(* Logix 5000 project; controller cal1632 1756-L62 rev 16.20; software revision 16.05; part 26 of 61 *)
(* tags used below, declared in another part *)
   AFI : BOOL;
   FAULT : BOOL;
   p01_param_turret_dia_ft : REAL;
   p01r02 : routine;
   p01r09_pb_global_reset : BOOL;
   p01r12_selected_line_speed : REAL;
   p01r13_line_running : BOOL;
   p01r13_line_slow_ramp : BOOL;
   p02_dint_from_hmi : hmi_dint;
   p11r31_timer_prs : TIMER;
   p13r03_hz : SYS_SCP;
   p13r30_request_cool : BOOL;
   p19_ai_prs : REAL;
   p19_di_pump : BOOL;
   p19_do_pump : BOOL;
   p19_param_zone_pressure : REAL;
   p19r30_request_cool : BOOL;
   p19r31 : routine;
   p19r31_pb_start : BOOL;
   p19r31_pb_stop : BOOL;
   p19r31_request_a00 : BOOL;
   p19r31_request_auto_run : BOOL;
   p19r31_request_manual_run : BOOL;
   p19r31_run_permissive : BOOL;
   p19r31_timer_fault : TIMER[4];
   p19r31_timer_warning : TIMER[4];
   p20_acc_fill_time_sec : REAL;
   p20_acc_input_max : REAL;
   p20_acc_input_min : REAL;
   p20_acc_output_max : REAL;
   p20_acc_output_min : REAL;
   p20_ai_acc_pstn : REAL;
   p20_ai_lc01 : REAL;
   p20_ai_letoff_dia : REAL;
   p20_ai_lo_turret_amps : REAL;
   p20_ai_lo_turret_hz : REAL;
   p20_ai_lo_turret_speed : REAL;
   p20_ai_loa_speed : REAL;
   p20_ai_lob_speed : REAL;
   p20_di_acc_door_open : BOOL;
   p20_di_acc_empty : BOOL;
   p20_di_acc_full : BOOL;
   p20_di_clutch_prs_ok : BOOL;
   p20_di_lfr_jog_fwd : BOOL;
   p20_di_lfr_jog_rev : BOOL;
   p20_di_lfr_nip_close : BOOL;
   p20_di_lo_turret : acs800_di_normal;
   p20_di_lo_turret_therm : BOOL;
   p20_di_loa_active : BOOL;
   p20_di_loa_brake : BOOL;
   p20_di_loa_fwd_dir : BOOL;
   p20_di_loa_jog : BOOL;
   p20_di_loa_start : BOOL;
   p20_di_loa_stop : BOOL;
   p20_di_loa_temp : BOOL;
   p20_di_lob_brake_thermostat : BOOL;
   p20_di_lob_fwd_dir : BOOL;
   p20_di_lob_jog : BOOL;
   p20_di_lob_motor_thermostat : BOOL;
   p20_di_lob_start : BOOL;
   p20_di_lob_stop : BOOL;
   p20_di_lof_acc_fill : BOOL;
   p20_di_turret_fwd : BOOL;
   p20_di_turret_pos : BOOL;
   p20_di_turret_rev : BOOL;
   p20_dia_input_max : REAL;
   p20_dia_input_min : REAL;
   p20_dia_output_max : REAL;
   p20_dia_output_min : REAL;
   p20_dint_to_hmi : DINT[16];
   p20_lc_input_max : REAL;
   p20_lc_input_min : REAL;
   p20_lc_output_max : REAL;
   p20_lc_output_min : REAL;
   p20_loa_ai_amps : REAL;
   p20_loa_ai_hz : REAL;
   p20_loa_ai_rpm : REAL;
   p20_loa_ai_torque : REAL;
   p20_loa_footage_input_max : REAL;
   p20_loa_footage_input_min : REAL;
   p20_loa_footage_output_max : REAL;
   p20_loa_footage_output_min : REAL;
   p20_lob_ai_amps : REAL;
   p20_lob_ai_hz : REAL;
   p20_lob_ai_rpm : REAL;
   p20_lob_ai_torque : REAL;
   p20_lob_footage_input_max : REAL;
   p20_lob_footage_input_min : REAL;
   p20_lob_footage_output_max : REAL;
   p20_lob_footage_output_min : REAL;
   p20_param_lo_turret_gear_ratio : REAL;
   p20_param_loa_gear_ratio : REAL;
   p20_param_lob_gear_ratio : REAL;
   p20_vfd_di_loa : acs800_di_normal;
   p20_vfd_di_lob : acs800_di_normal;
   p20r01 : routine;
   p20r02 : routine;
   p20r02_fault_exists : BOOL;
   p20r02_letoff_dia_ft : REAL;
   p20r02_letoff_selection_dwell : TIMER;
   p20r02_timer_fault : TIMER[4];
   p20r02_timer_warning : TIMER[4];
   p20r02_unack_fault : BOOL;
   p20r02_unack_warning : BOOL;
   p20r02_warning_exists : BOOL;
   p20r03 : routine;
   p20r03_accumulator_pct_scp : SYS_SCP;
   p20r03_accumulator_scp : SYS_SCP;
   p20r03_distance_to_core : REAL;
   p20r03_lo_radius : REAL;
   p20r03_lo_turret_speed_fb : SYS_RPM_TO_SPEED;
   p20r03_loa_distance_to_core : REAL;
   p20r03_Loa_footage_scp : SYS_SCP;
   p20r03_loa_speed_fb : SYS_RPM_TO_SPEED;
   p20r03_load_cell : SYS_SCP;
   p20r03_lob_distance_to_core : REAL;
   p20r03_Lob_footage_scp : SYS_SCP;
   p20r03_lob_speed_fb : SYS_RPM_TO_SPEED;
   p20r03_sensor_input : REAL;
   p20r03_sensor_scp : SYS_SCP;
   p20r03_timer_fault : TIMER[4];
   p20r03_timer_warning : TIMER[4];
   p20r04 : routine;
   p20r05 : routine;
   p20r06 : routine;
   p20r07 : routine;
   p20r08 : routine;
   p20r09 : routine;
   p20r10 : routine;
   p20r11 : routine;
   p20r13 : routine;
   p20r13_ai_acc_pct : REAL;
   p20r13_ai_loa_footage_ft : REAL;
   p20r13_ai_lob_footage_ft : REAL;
   p20r14 : routine;
   p20r15 : routine;
   p20r15_loa_on : BOOL;
   p20r16 : routine;
   p20r16_lob_on : BOOL;
   p20r17 : routine;
   p20r17_letoff_avg_diam_inch : REAL;
   p20r18 : routine;
   p22_ao_selected_speed : REAL;
(* P19_Advanced_Cooling, continued *)

ROUTINE R31_Pump   (* ladder *)
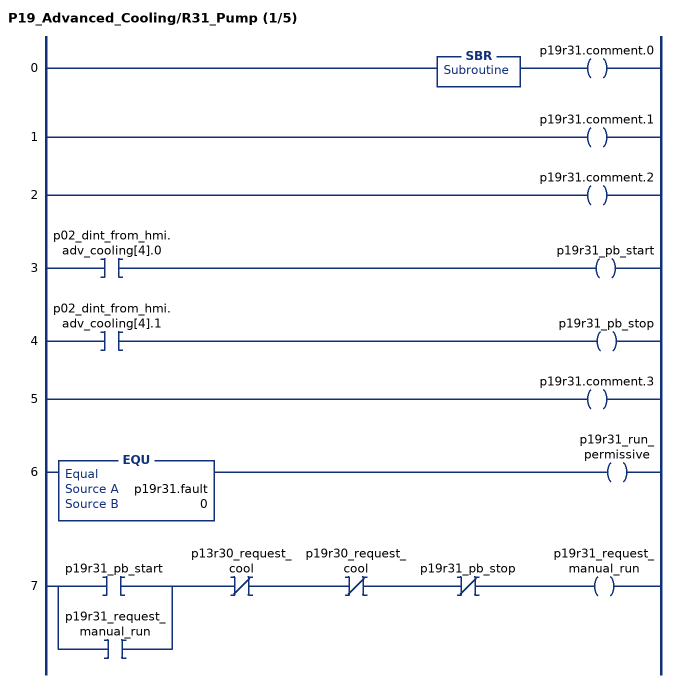
   0: SBR()OTE(p19r31.comment.0);
   1: OTE(p19r31.comment.1);
   2: OTE(p19r31.comment.2);
   3: XIC(p02_dint_from_hmi.adv_cooling[4].0)OTE(p19r31_pb_start);
   4: XIC(p02_dint_from_hmi.adv_cooling[4].1)OTE(p19r31_pb_stop);
   5: OTE(p19r31.comment.3);
   6: EQU(p19r31.fault,0)OTE(p19r31_run_permissive);
   7: [XIC(p19r31_pb_start) ,XIC(p19r31_request_manual_run) ]XIO(p13r30_request_cool)XIO(p19r30_request_cool)XIO(p19r31_pb_stop)OTE(p19r31_request_manual_run);
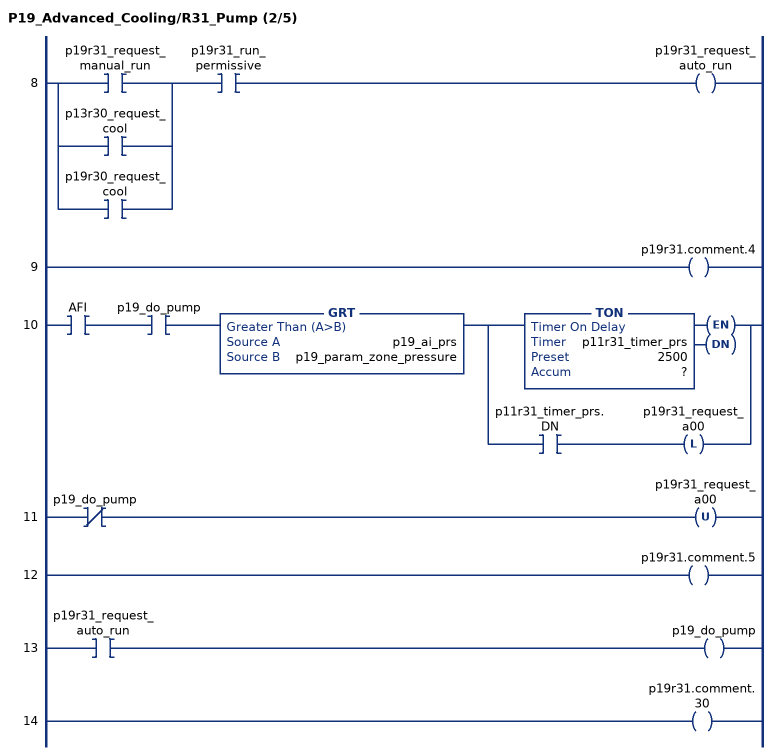
   8: [XIC(p19r31_request_manual_run) ,XIC(p13r30_request_cool) ,XIC(p19r30_request_cool) ]XIC(p19r31_run_permissive)OTE(p19r31_request_auto_run);
   9: OTE(p19r31.comment.4);
   10: XIC(AFI)XIC(p19_do_pump)GRT(p19_ai_prs,p19_param_zone_pressure)[TON(p11r31_timer_prs,?,?) ,XIC(p11r31_timer_prs.DN) OTL(p19r31_request_a00) ];
   11: XIO(p19_do_pump)OTU(p19r31_request_a00);
   12: OTE(p19r31.comment.5);
   13: XIC(p19r31_request_auto_run)OTE(p19_do_pump);
   14: OTE(p19r31.comment.30);
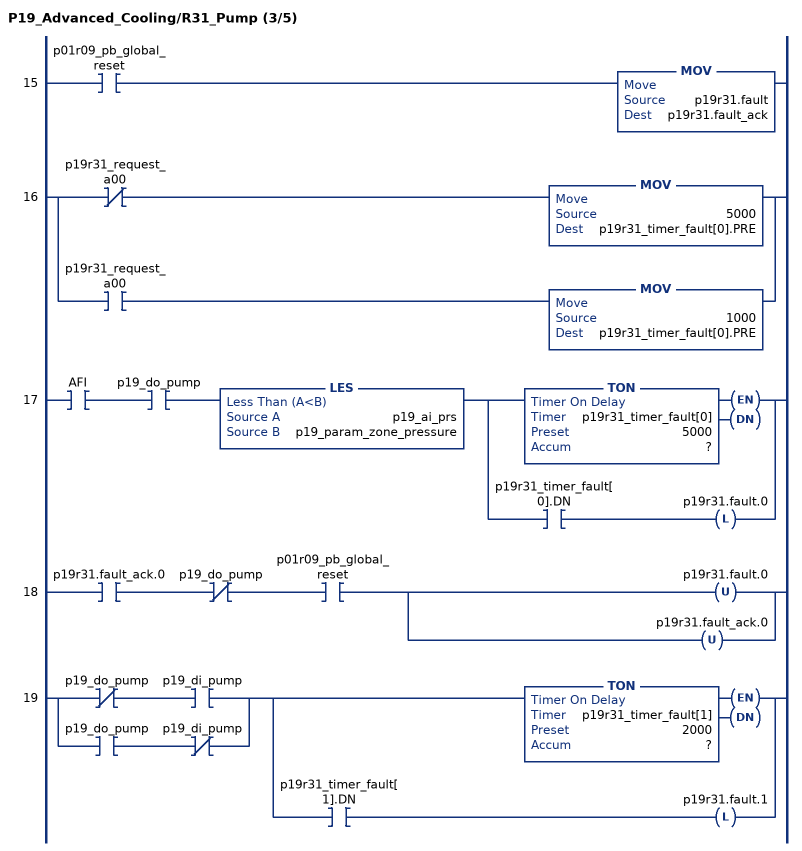
   15: XIC(p01r09_pb_global_reset)MOV(p19r31.fault,p19r31.fault_ack);
   16: [XIO(p19r31_request_a00) MOV(5000,p19r31_timer_fault[0].PRE) ,XIC(p19r31_request_a00) MOV(1000,p19r31_timer_fault[0].PRE) ];
   17: XIC(AFI)XIC(p19_do_pump)LES(p19_ai_prs,p19_param_zone_pressure)[TON(p19r31_timer_fault[0],?,?) ,XIC(p19r31_timer_fault[0].DN) OTL(p19r31.fault.0) ];
   18: XIC(p19r31.fault_ack.0)XIO(p19_do_pump)XIC(p01r09_pb_global_reset)[OTU(p19r31.fault.0) ,OTU(p19r31.fault_ack.0) ];
   19: [XIO(p19_do_pump) XIC(p19_di_pump) ,XIC(p19_do_pump) XIO(p19_di_pump) ][TON(p19r31_timer_fault[1],?,?) ,XIC(p19r31_timer_fault[1].DN) OTL(p19r31.fault.1) ];
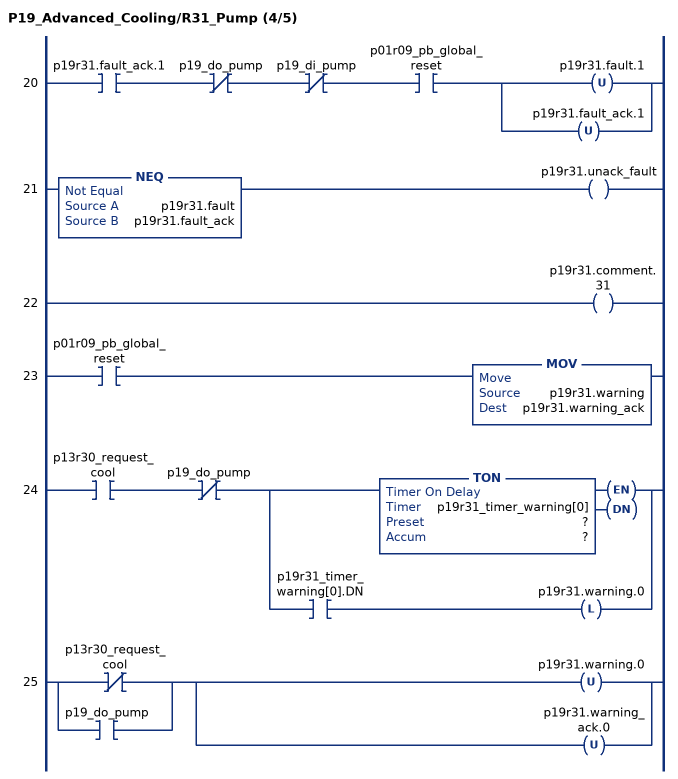
   20: XIC(p19r31.fault_ack.1)XIO(p19_do_pump)XIO(p19_di_pump)XIC(p01r09_pb_global_reset)[OTU(p19r31.fault.1) ,OTU(p19r31.fault_ack.1) ];
   21: NEQ(p19r31.fault,p19r31.fault_ack)OTE(p19r31.unack_fault);
   22: OTE(p19r31.comment.31);
   23: XIC(p01r09_pb_global_reset)MOV(p19r31.warning,p19r31.warning_ack);
   24: XIC(p13r30_request_cool)XIO(p19_do_pump)[TON(p19r31_timer_warning[0],?,?) ,XIC(p19r31_timer_warning[0].DN) OTL(p19r31.warning.0) ];
   25: [XIO(p13r30_request_cool) ,XIC(p19_do_pump) ][OTU(p19r31.warning.0) ,OTU(p19r31.warning_ack.0) ];
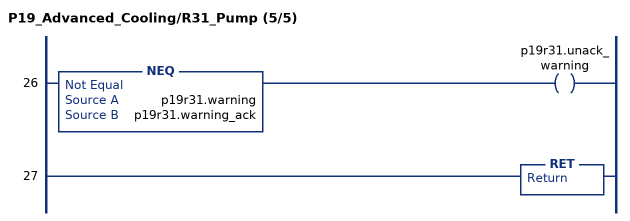
   26: NEQ(p19r31.warning,p19r31.warning_ack)OTE(p19r31.unack_warning);
   27: RET();
END_ROUTINE
END_PROGRAM

PROGRAM P20_Letoff   (* main routine R01_Main *)

ROUTINE R01_Main   (* ladder *)
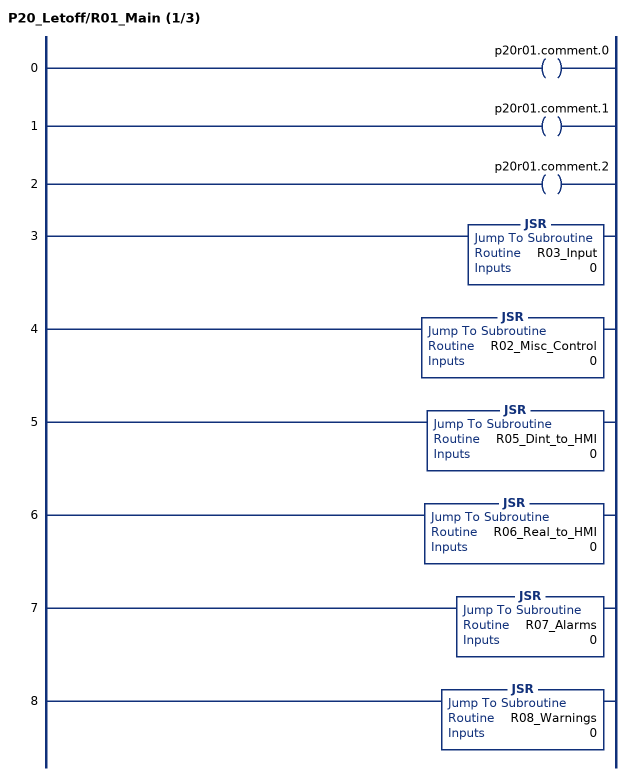
   0: OTE(p20r01.comment.0);
   1: OTE(p20r01.comment.1);
   2: OTE(p20r01.comment.2);
   3: JSR(R03_Input,0);
   4: JSR(R02_Misc_Control,0);
   5: JSR(R05_Dint_to_HMI,0);
   6: JSR(R06_Real_to_HMI,0);
   7: JSR(R07_Alarms,0);
   8: JSR(R08_Warnings,0);
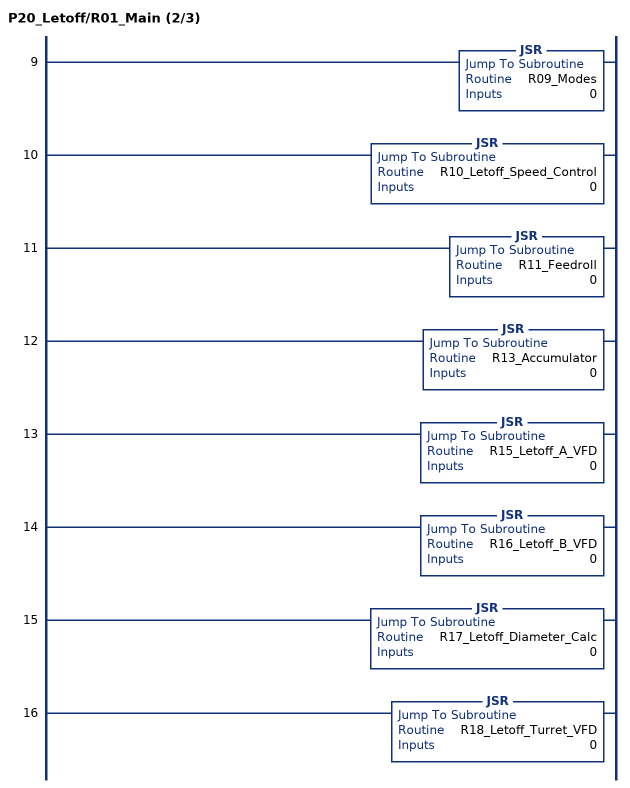
   9: JSR(R09_Modes,0);
   10: JSR(R10_Letoff_Speed_Control,0);
   11: JSR(R11_Feedroll,0);
   12: JSR(R13_Accumulator,0);
   13: JSR(R15_Letoff_A_VFD,0);
   14: JSR(R16_Letoff_B_VFD,0);
   15: JSR(R17_Letoff_Diameter_Calc,0);
   16: JSR(R18_Letoff_Turret_VFD,0);
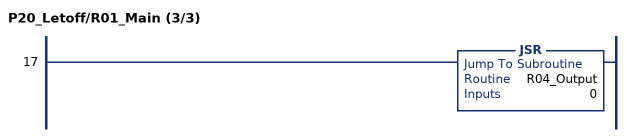
   17: JSR(R04_Output,0);
END_ROUTINE

ROUTINE R02_Misc_Control   (* ladder *)
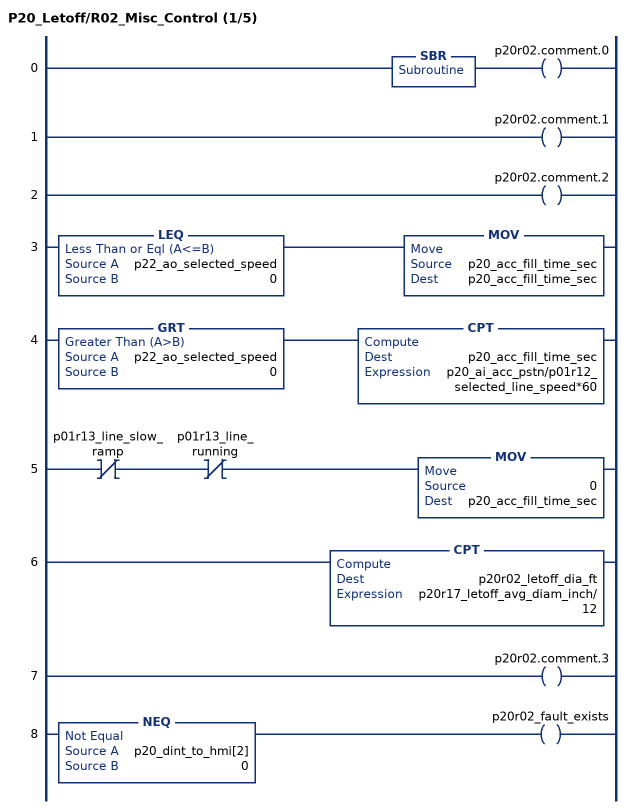
   0: SBR()OTE(p20r02.comment.0);
   1: OTE(p20r02.comment.1);
   2: OTE(p20r02.comment.2);
   3: LEQ(p22_ao_selected_speed,0)MOV(p20_acc_fill_time_sec,p20_acc_fill_time_sec);
   4: GRT(p22_ao_selected_speed,0)CPT(p20_acc_fill_time_sec,p20_ai_acc_pstn/p01r12_selected_line_speed*60);
   5: XIO(p01r13_line_slow_ramp)XIO(p01r13_line_running)MOV(0,p20_acc_fill_time_sec);
   6: CPT(p20r02_letoff_dia_ft,p20r17_letoff_avg_diam_inch/12);
   7: OTE(p20r02.comment.3);
   8: NEQ(p20_dint_to_hmi[2],0)OTE(p20r02_fault_exists);
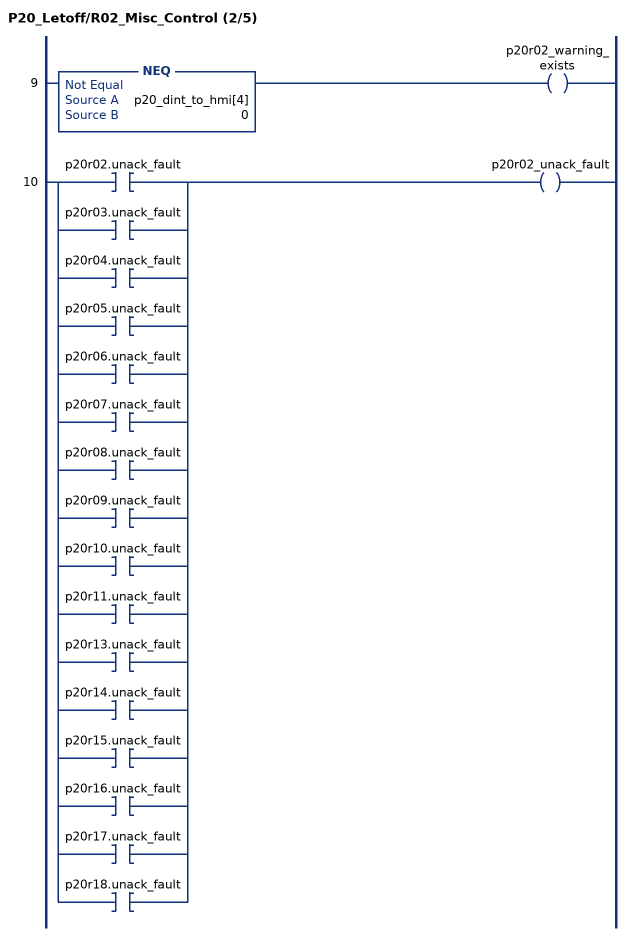
   9: NEQ(p20_dint_to_hmi[4],0)OTE(p20r02_warning_exists);
   10: [XIC(p20r02.unack_fault) ,XIC(p20r03.unack_fault) ,XIC(p20r04.unack_fault) ,XIC(p20r05.unack_fault) ,XIC(p20r06.unack_fault) ,XIC(p20r07.unack_fault) ,XIC(p20r08.unack_fault) ,XIC(p20r09.unack_fault) ,XIC(p20r10.unack_fault) ,XIC(p20r11.unack_fault) ,XIC(p20r13.unack_fault) ,XIC(p20r14.unack_fault) ,XIC(p20r15.unack_fault) ,XIC(p20r16.unack_fault) ,XIC(p20r17.unack_fault) ,XIC(p20r18.unack_fault) ]OTE(p20r02_unack_fault);
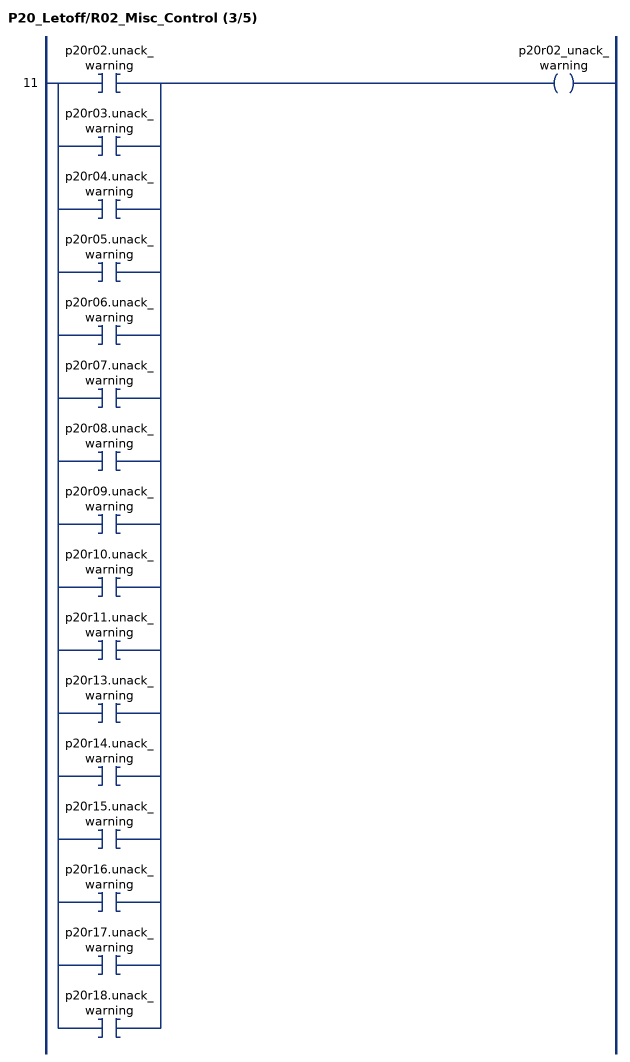
   11: [XIC(p20r02.unack_warning) ,XIC(p20r03.unack_warning) ,XIC(p20r04.unack_warning) ,XIC(p20r05.unack_warning) ,XIC(p20r06.unack_warning) ,XIC(p20r07.unack_warning) ,XIC(p20r08.unack_warning) ,XIC(p20r09.unack_warning) ,XIC(p20r10.unack_warning) ,XIC(p20r11.unack_warning) ,XIC(p20r13.unack_warning) ,XIC(p20r14.unack_warning) ,XIC(p20r15.unack_warning) ,XIC(p20r16.unack_warning) ,XIC(p20r17.unack_warning) ,XIC(p20r18.unack_warning) ]OTE(p20r02_unack_warning);
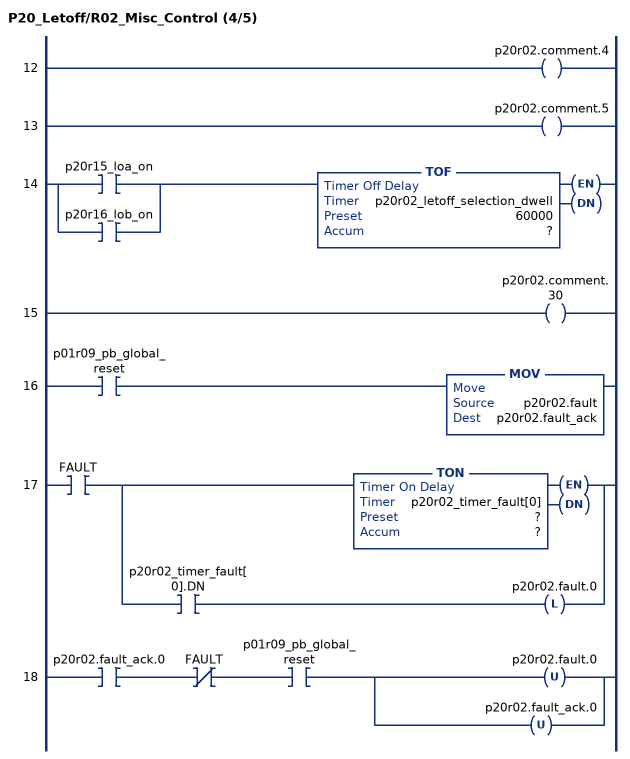
   12: OTE(p20r02.comment.4);
   13: OTE(p20r02.comment.5);
   14: [XIC(p20r15_loa_on) ,XIC(p20r16_lob_on) ]TOF(p20r02_letoff_selection_dwell,?,?);
   15: OTE(p20r02.comment.30);
   16: XIC(p01r09_pb_global_reset)MOV(p20r02.fault,p20r02.fault_ack);
   17: XIC(FAULT)[TON(p20r02_timer_fault[0],?,?) ,XIC(p20r02_timer_fault[0].DN) OTL(p20r02.fault.0) ];
   18: XIC(p20r02.fault_ack.0)XIO(FAULT)XIC(p01r09_pb_global_reset)[OTU(p20r02.fault.0) ,OTU(p20r02.fault_ack.0) ];
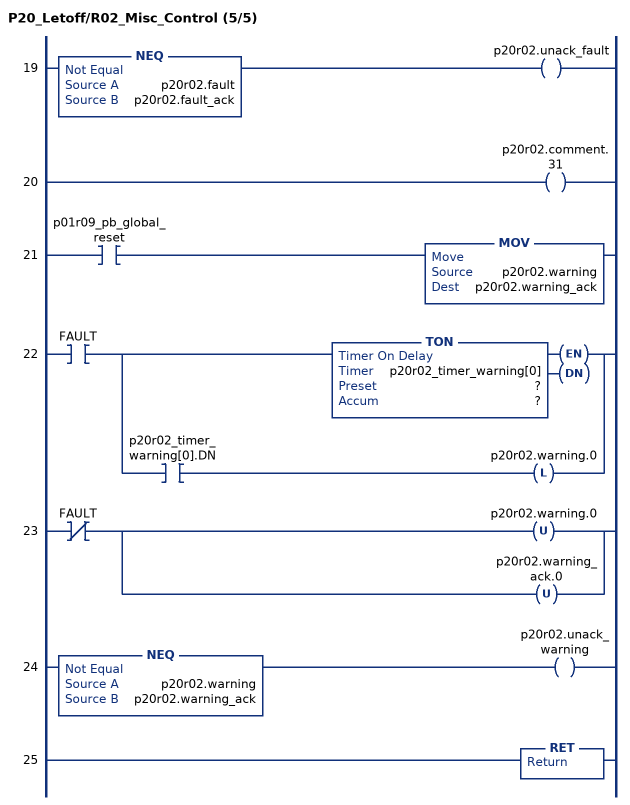
   19: NEQ(p20r02.fault,p20r02.fault_ack)OTE(p20r02.unack_fault);
   20: OTE(p20r02.comment.31);
   21: XIC(p01r09_pb_global_reset)MOV(p20r02.warning,p20r02.warning_ack);
   22: XIC(FAULT)[TON(p20r02_timer_warning[0],?,?) ,XIC(p20r02_timer_warning[0].DN) OTL(p20r02.warning.0) ];
   23: XIO(FAULT)[OTU(p20r02.warning.0) ,OTU(p20r02.warning_ack.0) ];
   24: NEQ(p20r02.warning,p20r02.warning_ack)OTE(p20r02.unack_warning);
   25: RET();
END_ROUTINE

ROUTINE R03_Input   (* ladder *)
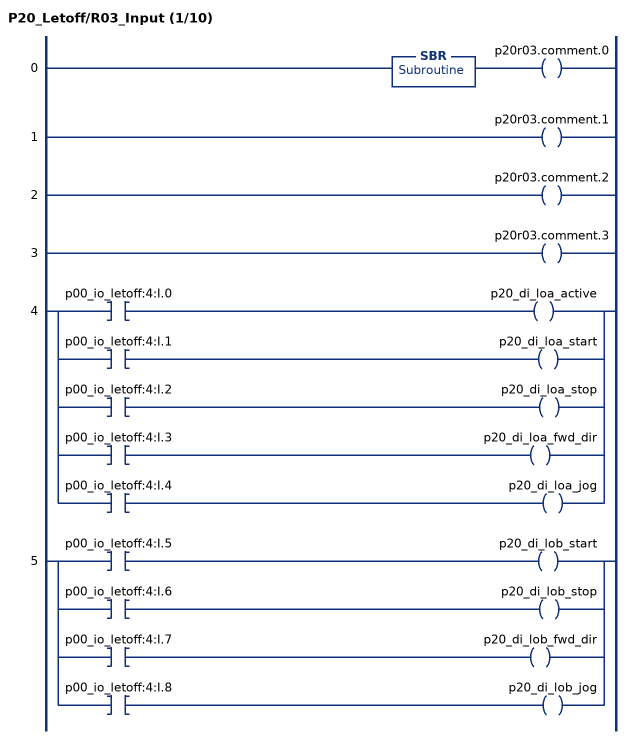
   0: SBR()OTE(p20r03.comment.0);
   1: OTE(p20r03.comment.1);
   2: OTE(p20r03.comment.2);
   3: OTE(p20r03.comment.3);
   4: [XIC(p00_io_letoff:4:I.0) OTE(p20_di_loa_active) ,XIC(p00_io_letoff:4:I.1) OTE(p20_di_loa_start) ,XIC(p00_io_letoff:4:I.2) OTE(p20_di_loa_stop) ,XIC(p00_io_letoff:4:I.3) OTE(p20_di_loa_fwd_dir) ,XIC(p00_io_letoff:4:I.4) OTE(p20_di_loa_jog) ];
   5: [XIC(p00_io_letoff:4:I.5) OTE(p20_di_lob_start) ,XIC(p00_io_letoff:4:I.6) OTE(p20_di_lob_stop) ,XIC(p00_io_letoff:4:I.7) OTE(p20_di_lob_fwd_dir) ,XIC(p00_io_letoff:4:I.8) OTE(p20_di_lob_jog) ];
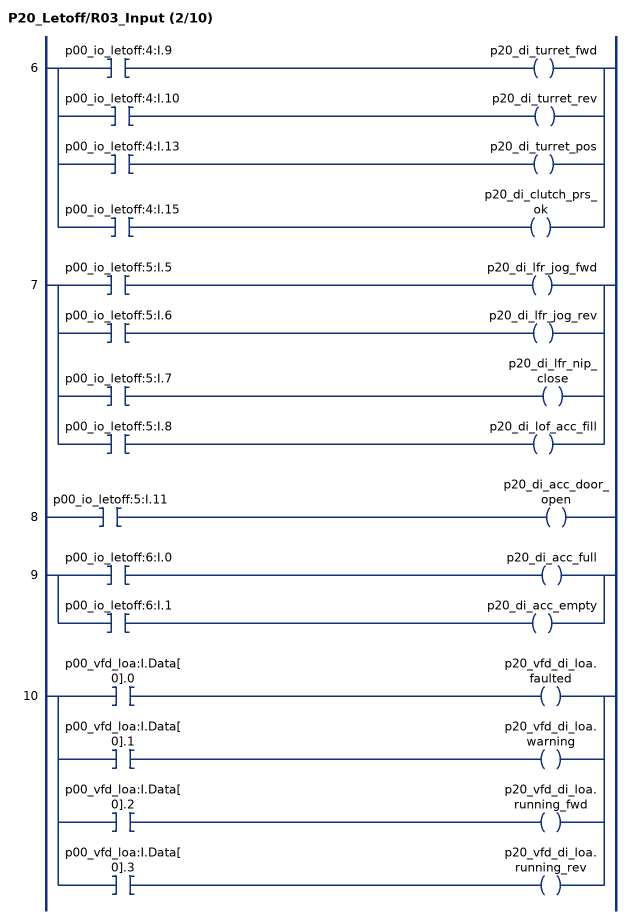
   6: [XIC(p00_io_letoff:4:I.9) OTE(p20_di_turret_fwd) ,XIC(p00_io_letoff:4:I.10) OTE(p20_di_turret_rev) ,XIC(p00_io_letoff:4:I.13) OTE(p20_di_turret_pos) ,XIC(p00_io_letoff:4:I.15) OTE(p20_di_clutch_prs_ok) ];
   7: [XIC(p00_io_letoff:5:I.5) OTE(p20_di_lfr_jog_fwd) ,XIC(p00_io_letoff:5:I.6) OTE(p20_di_lfr_jog_rev) ,XIC(p00_io_letoff:5:I.7) OTE(p20_di_lfr_nip_close) ,XIC(p00_io_letoff:5:I.8) OTE(p20_di_lof_acc_fill) ];
   8: XIC(p00_io_letoff:5:I.11)OTE(p20_di_acc_door_open);
   9: [XIC(p00_io_letoff:6:I.0) OTE(p20_di_acc_full) ,XIC(p00_io_letoff:6:I.1) OTE(p20_di_acc_empty) ];
   10: [XIC(p00_vfd_loa:I.Data[0].0) OTE(p20_vfd_di_loa.faulted) ,XIC(p00_vfd_loa:I.Data[0].1) OTE(p20_vfd_di_loa.warning) ,XIC(p00_vfd_loa:I.Data[0].2) OTE(p20_vfd_di_loa.running_fwd) ,XIC(p00_vfd_loa:I.Data[0].3) OTE(p20_vfd_di_loa.running_rev) ];
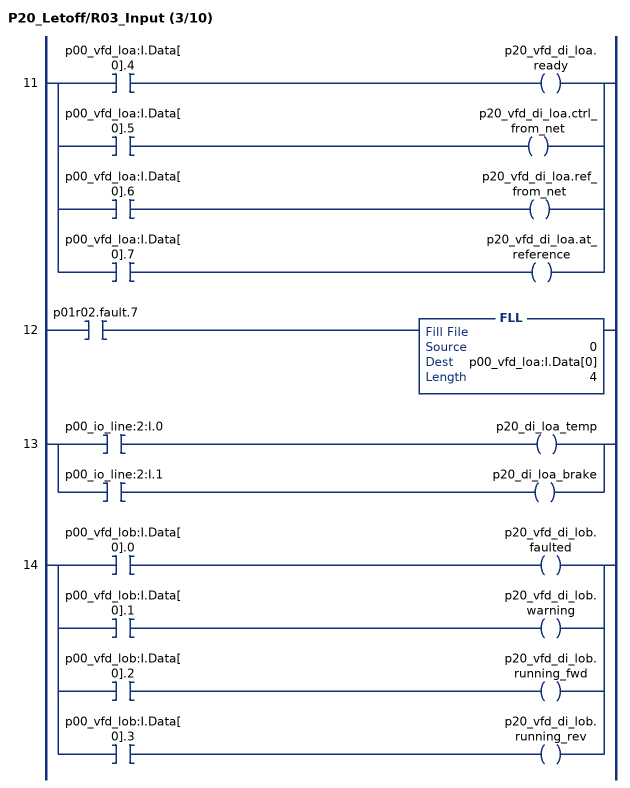
   11: [XIC(p00_vfd_loa:I.Data[0].4) OTE(p20_vfd_di_loa.ready) ,XIC(p00_vfd_loa:I.Data[0].5) OTE(p20_vfd_di_loa.ctrl_from_net) ,XIC(p00_vfd_loa:I.Data[0].6) OTE(p20_vfd_di_loa.ref_from_net) ,XIC(p00_vfd_loa:I.Data[0].7) OTE(p20_vfd_di_loa.at_reference) ];
   12: XIC(p01r02.fault.7)FLL(0,p00_vfd_loa:I.Data[0],4);
   13: [XIC(p00_io_line:2:I.0) OTE(p20_di_loa_temp) ,XIC(p00_io_line:2:I.1) OTE(p20_di_loa_brake) ];
   14: [XIC(p00_vfd_lob:I.Data[0].0) OTE(p20_vfd_di_lob.faulted) ,XIC(p00_vfd_lob:I.Data[0].1) OTE(p20_vfd_di_lob.warning) ,XIC(p00_vfd_lob:I.Data[0].2) OTE(p20_vfd_di_lob.running_fwd) ,XIC(p00_vfd_lob:I.Data[0].3) OTE(p20_vfd_di_lob.running_rev) ];
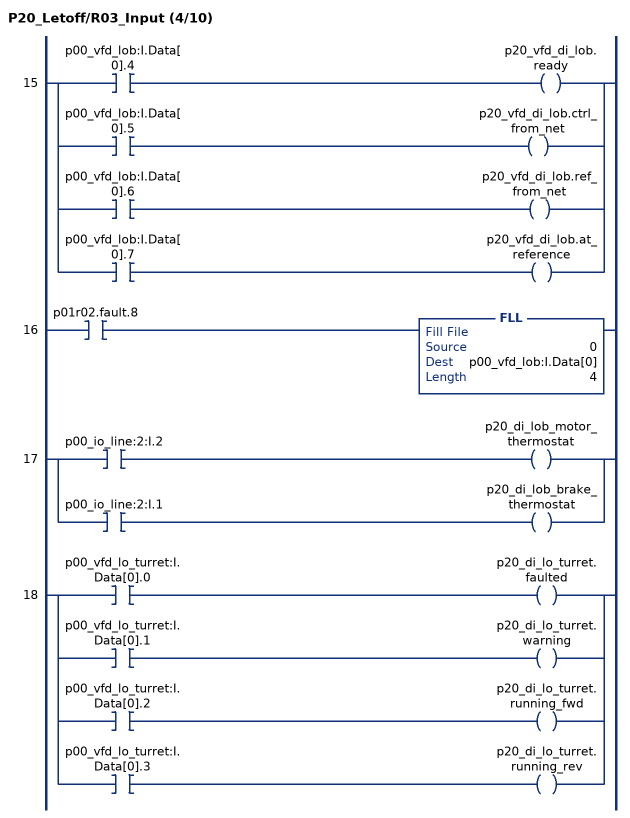
   15: [XIC(p00_vfd_lob:I.Data[0].4) OTE(p20_vfd_di_lob.ready) ,XIC(p00_vfd_lob:I.Data[0].5) OTE(p20_vfd_di_lob.ctrl_from_net) ,XIC(p00_vfd_lob:I.Data[0].6) OTE(p20_vfd_di_lob.ref_from_net) ,XIC(p00_vfd_lob:I.Data[0].7) OTE(p20_vfd_di_lob.at_reference) ];
   16: XIC(p01r02.fault.8)FLL(0,p00_vfd_lob:I.Data[0],4);
   17: [XIC(p00_io_line:2:I.2) OTE(p20_di_lob_motor_thermostat) ,XIC(p00_io_line:2:I.1) OTE(p20_di_lob_brake_thermostat) ];
   18: [XIC(p00_vfd_lo_turret:I.Data[0].0) OTE(p20_di_lo_turret.faulted) ,XIC(p00_vfd_lo_turret:I.Data[0].1) OTE(p20_di_lo_turret.warning) ,XIC(p00_vfd_lo_turret:I.Data[0].2) OTE(p20_di_lo_turret.running_fwd) ,XIC(p00_vfd_lo_turret:I.Data[0].3) OTE(p20_di_lo_turret.running_rev) ];
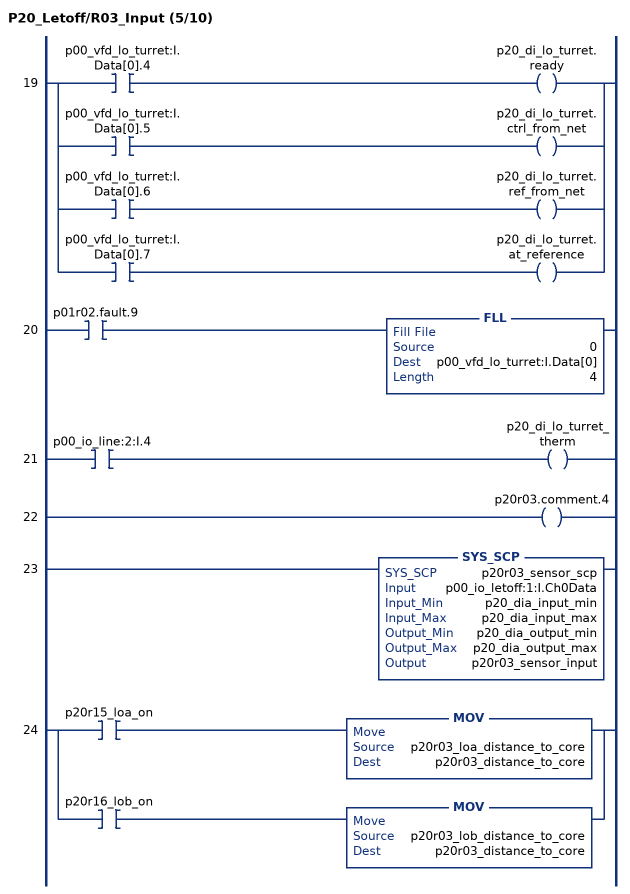
   19: [XIC(p00_vfd_lo_turret:I.Data[0].4) OTE(p20_di_lo_turret.ready) ,XIC(p00_vfd_lo_turret:I.Data[0].5) OTE(p20_di_lo_turret.ctrl_from_net) ,XIC(p00_vfd_lo_turret:I.Data[0].6) OTE(p20_di_lo_turret.ref_from_net) ,XIC(p00_vfd_lo_turret:I.Data[0].7) OTE(p20_di_lo_turret.at_reference) ];
   20: XIC(p01r02.fault.9)FLL(0,p00_vfd_lo_turret:I.Data[0],4);
   21: XIC(p00_io_line:2:I.4)OTE(p20_di_lo_turret_therm);
   22: OTE(p20r03.comment.4);
   23: SYS_SCP(p20r03_sensor_scp,p00_io_letoff:1:I.Ch0Data,p20_dia_input_min,p20_dia_input_max,p20_dia_output_min,p20_dia_output_max,p20r03_sensor_input);
   24: [XIC(p20r15_loa_on) MOV(p20r03_loa_distance_to_core,p20r03_distance_to_core) ,XIC(p20r16_lob_on) MOV(p20r03_lob_distance_to_core,p20r03_distance_to_core) ];
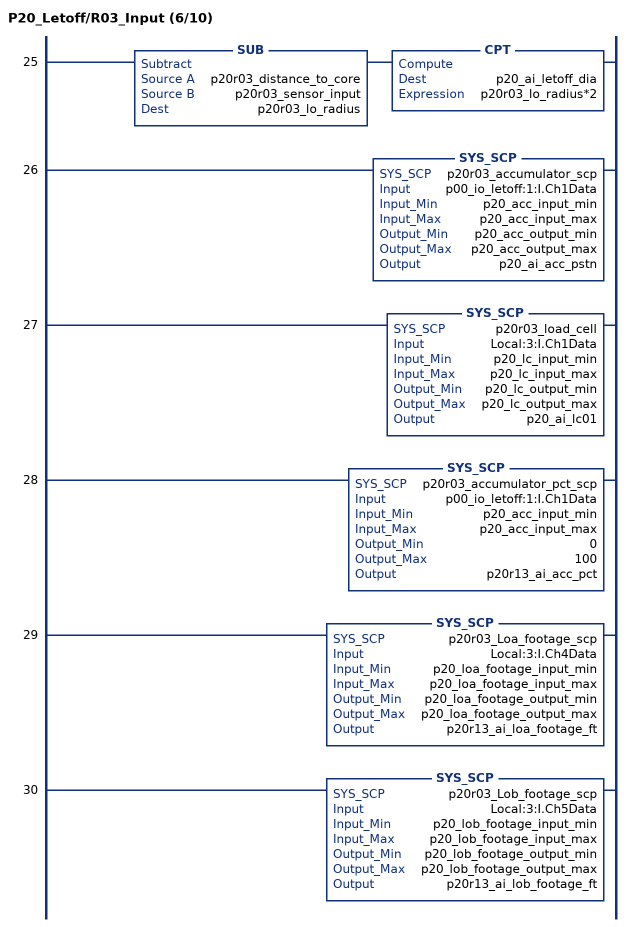
   25: SUB(p20r03_distance_to_core,p20r03_sensor_input,p20r03_lo_radius)CPT(p20_ai_letoff_dia,p20r03_lo_radius*2);
   26: SYS_SCP(p20r03_accumulator_scp,p00_io_letoff:1:I.Ch1Data,p20_acc_input_min,p20_acc_input_max,p20_acc_output_min,p20_acc_output_max,p20_ai_acc_pstn);
   27: SYS_SCP(p20r03_load_cell,Local:3:I.Ch1Data,p20_lc_input_min,p20_lc_input_max,p20_lc_output_min,p20_lc_output_max,p20_ai_lc01);
   28: SYS_SCP(p20r03_accumulator_pct_scp,p00_io_letoff:1:I.Ch1Data,p20_acc_input_min,p20_acc_input_max,0,100,p20r13_ai_acc_pct);
   29: SYS_SCP(p20r03_Loa_footage_scp,Local:3:I.Ch4Data,p20_loa_footage_input_min,p20_loa_footage_input_max,p20_loa_footage_output_min,p20_loa_footage_output_max,p20r13_ai_loa_footage_ft);
   30: SYS_SCP(p20r03_Lob_footage_scp,Local:3:I.Ch5Data,p20_lob_footage_input_min,p20_lob_footage_input_max,p20_lob_footage_output_min,p20_lob_footage_output_max,p20r13_ai_lob_footage_ft);
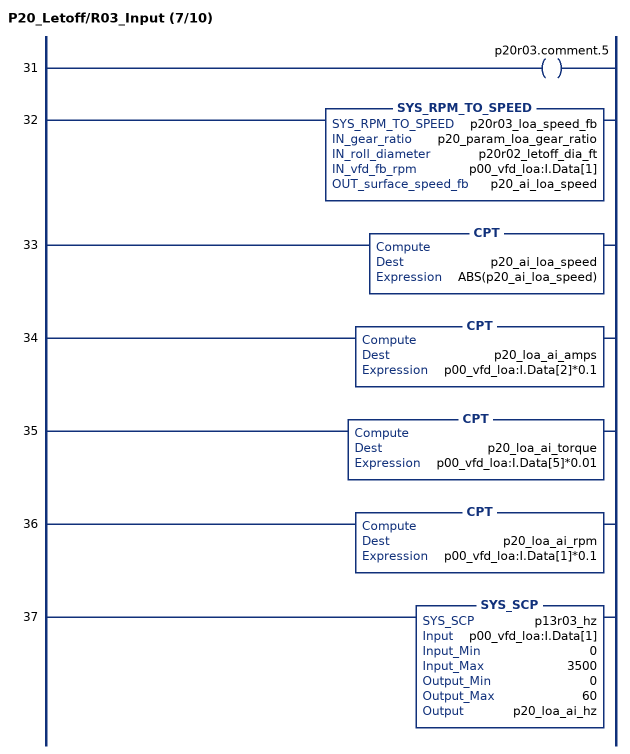
   31: OTE(p20r03.comment.5);
   32: SYS_RPM_TO_SPEED(p20r03_loa_speed_fb,p20_param_loa_gear_ratio,p20r02_letoff_dia_ft,p00_vfd_loa:I.Data[1],p20_ai_loa_speed);
   33: CPT(p20_ai_loa_speed,ABS(p20_ai_loa_speed));
   34: CPT(p20_loa_ai_amps,p00_vfd_loa:I.Data[2]*0.1);
   35: CPT(p20_loa_ai_torque,p00_vfd_loa:I.Data[5]*0.01);
   36: CPT(p20_loa_ai_rpm,p00_vfd_loa:I.Data[1]*0.1);
   37: SYS_SCP(p13r03_hz,p00_vfd_loa:I.Data[1],0,3500,0,60,p20_loa_ai_hz);
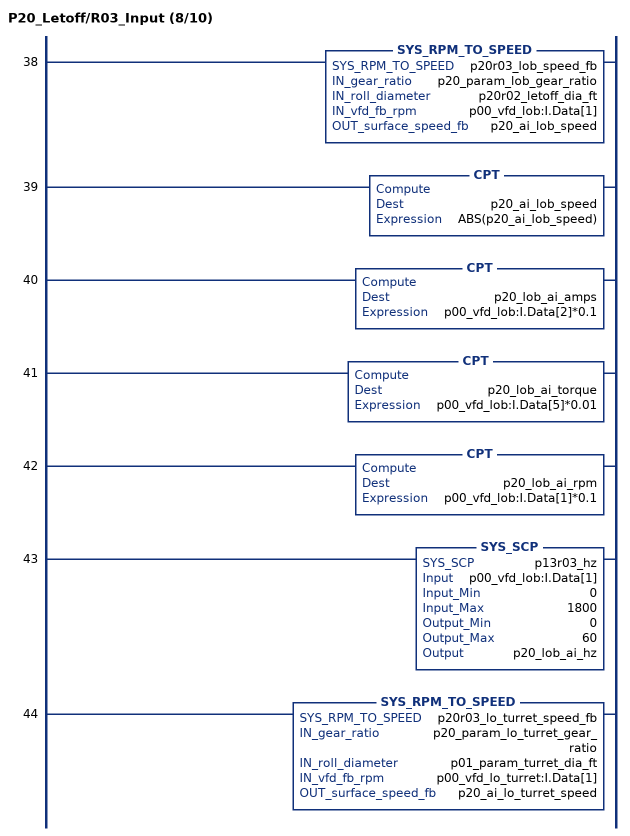
   38: SYS_RPM_TO_SPEED(p20r03_lob_speed_fb,p20_param_lob_gear_ratio,p20r02_letoff_dia_ft,p00_vfd_lob:I.Data[1],p20_ai_lob_speed);
   39: CPT(p20_ai_lob_speed,ABS(p20_ai_lob_speed));
   40: CPT(p20_lob_ai_amps,p00_vfd_lob:I.Data[2]*0.1);
   41: CPT(p20_lob_ai_torque,p00_vfd_lob:I.Data[5]*0.01);
   42: CPT(p20_lob_ai_rpm,p00_vfd_lob:I.Data[1]*0.1);
   43: SYS_SCP(p13r03_hz,p00_vfd_lob:I.Data[1],0,1800,0,60,p20_lob_ai_hz);
   44: SYS_RPM_TO_SPEED(p20r03_lo_turret_speed_fb,p20_param_lo_turret_gear_ratio,p01_param_turret_dia_ft,p00_vfd_lo_turret:I.Data[1],p20_ai_lo_turret_speed);
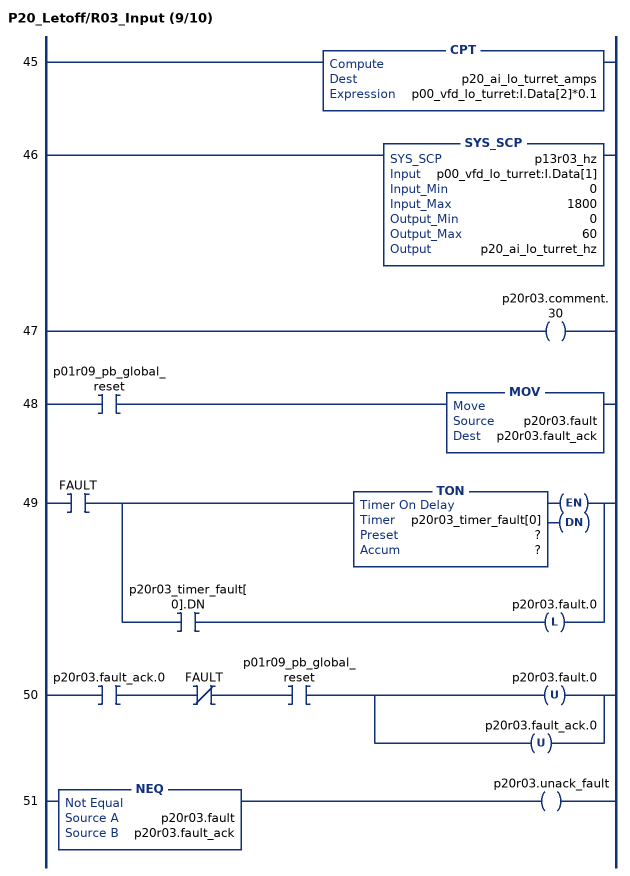
   45: CPT(p20_ai_lo_turret_amps,p00_vfd_lo_turret:I.Data[2]*0.1);
   46: SYS_SCP(p13r03_hz,p00_vfd_lo_turret:I.Data[1],0,1800,0,60,p20_ai_lo_turret_hz);
   47: OTE(p20r03.comment.30);
   48: XIC(p01r09_pb_global_reset)MOV(p20r03.fault,p20r03.fault_ack);
   49: XIC(FAULT)[TON(p20r03_timer_fault[0],?,?) ,XIC(p20r03_timer_fault[0].DN) OTL(p20r03.fault.0) ];
   50: XIC(p20r03.fault_ack.0)XIO(FAULT)XIC(p01r09_pb_global_reset)[OTU(p20r03.fault.0) ,OTU(p20r03.fault_ack.0) ];
   51: NEQ(p20r03.fault,p20r03.fault_ack)OTE(p20r03.unack_fault);
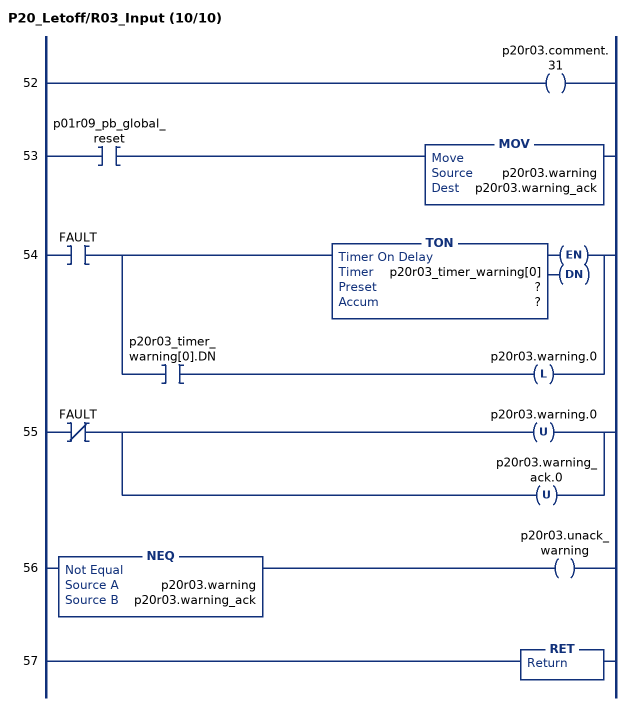
   52: OTE(p20r03.comment.31);
   53: XIC(p01r09_pb_global_reset)MOV(p20r03.warning,p20r03.warning_ack);
   54: XIC(FAULT)[TON(p20r03_timer_warning[0],?,?) ,XIC(p20r03_timer_warning[0].DN) OTL(p20r03.warning.0) ];
   55: XIO(FAULT)[OTU(p20r03.warning.0) ,OTU(p20r03.warning_ack.0) ];
   56: NEQ(p20r03.warning,p20r03.warning_ack)OTE(p20r03.unack_warning);
   57: RET();
END_ROUTINE
